{attribute 'linkalways'} 
{attribute 'no_explicit_call' := 'This FB is a CLASS and must be accessed using methods or properties'}
{attribute 'enable_dynamic_creation'}
FUNCTION_BLOCK ArrayDatatypeAddedEvent EXTENDS Disposable IMPLEMENTS I_ArrayDatatypeAddedEvent
VAR
	_target : I_ArrayDatatype;
END_VAR

METHOD FB_init : BOOL
VAR_INPUT
	bInitRetains : BOOL; // if TRUE, the retain variables are initialized (warm start / cold start)
	bInCopyCode : BOOL;  // if TRUE, the instance afterwards gets moved into the copy code (online change)
	Target : I_ArrayDatatype;
END_VAR
This^._target := Target;
END_METHOD

PROPERTY PUBLIC Target : I_ArrayDatatype
GET
Target := _target;
END_GET
END_PROPERTY

END_FUNCTION_BLOCK

(* stored: Version 1.1.0.1, ProductVersion 3.1.4024.13
   POU ArrayDatatypeAddedEvent: Id {d70d9279-c19b-0f54-0966-ce94b449e283}, SpecialFunc None
   Folder Constructor: Id {f042406a-c67e-0780-2b6d-90bea288b108}
   Method FB_init: Id {45f7dec8-fd28-0646-186c-65f9dec329e7}
   Property Target: Id {c0b629ba-30ca-0d40-2839-1240d8c9bb87}
   Get Get: Id {58c540ff-0f0b-0b14-2650-ee49bff8d3f3} *)
